// Mitsubishi GX Works2 project: PLC 특수기능 (Falling Pulse 예제)   PLC: Q03UDV

PROGRAM MAIN
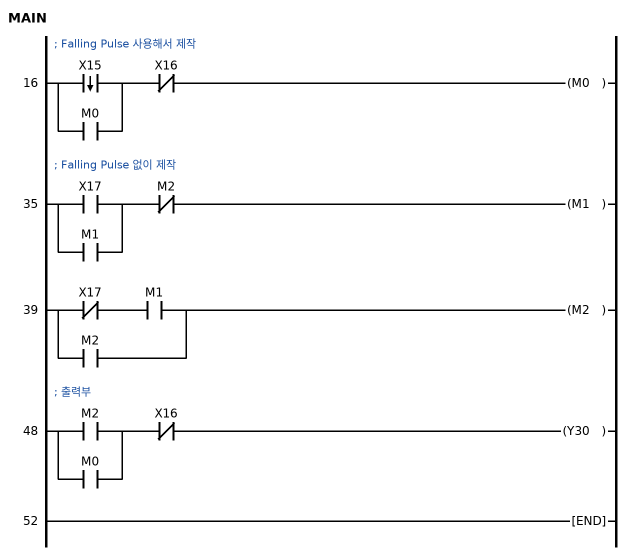
; Falling Pulse 사용해서 제작
16    LDF     X15
      OR      M0
      ANI     X16
      OUT     M0
; Falling Pulse 없이 제작
35    LD      X17
      OR      M1
      ANI     M2
      OUT     M1
39    LDI     X17
      AND     M1
      OR      M2
      OUT     M2
; 출력부
48    LD      M2
      OR      M0
      ANI     X16
      OUT     Y30
52    END
END_PROGRAM
